# B&R Automation Studio project BRLAB12
Automation Studio 4.5.2.102

## Configuration Config1

### Task classes (Cpu.sw)
```
Cyclic#1:
  Program <- Program.prg
Binaries: udbdef, TCData, ashwd, User, asfw, arconfig, sysconf, Role, ashwac, iomap
Libraries: MotorCtrl
```

### Hardware
```
4PP065_0571_P74 : 4PP065.0571-P74 v1.1.2.0
  Connector IF5:
    ActivateDevice = 1
  ConfigurationID = firstblood_Config1
  Simulation = 1
```

## Logical view

### Library Logical/Libraries/MotorCtrl (ANSIC)

#### MotorCtrl.fun - Exported functions and function blocks
```iecst
{REDUND_ERROR} FUNCTION_BLOCK FB_Controller (*TODO: Add your comment here*) (*$GROUP=User,$CAT=User,$GROUPICON=User.png,$CATICON=User.png*)
	VAR_INPUT
		e : REAL;
	END_VAR
	VAR_OUTPUT
		u : REAL;
	END_VAR
	VAR
		k_p : REAL;
		k_i : REAL;
		iyOld : REAL;
		max_abs_value : REAL;
		dt : REAL;
		integrator : FB_Integrator;
	END_VAR
END_FUNCTION_BLOCK

{REDUND_ERROR} FUNCTION_BLOCK FB_Integrator (*TODO: Add your comment here*) (*$GROUP=User,$CAT=User,$GROUPICON=User.png,$CATICON=User.png*)
	VAR_INPUT
		in : REAL;
	END_VAR
	VAR_OUTPUT
		out : REAL;
	END_VAR
	VAR
		dt : REAL;
		temp : REAL;
	END_VAR
END_FUNCTION_BLOCK

{REDUND_ERROR} FUNCTION_BLOCK FB_Motor (*TODO: Add your comment here*) (*$GROUP=User,$CAT=User,$GROUPICON=User.png,$CATICON=User.png*)
	VAR_INPUT
		u : REAL;
	END_VAR
	VAR_OUTPUT
		w : REAL;
		phi : REAL;
	END_VAR
	VAR
		integrator1 : FB_Integrator;
		integrator2 : FB_Integrator;
		Tm : REAL;
		ke : REAL;
		dt : REAL;
	END_VAR
END_FUNCTION_BLOCK
```

#### FB_Controller.c
```c
#include <bur/plctypes.h>
#ifdef __cplusplus
	extern "C"
	{
#endif
	#include "MotorCtrl.h"
#ifdef __cplusplus
	};
#endif

void FB_Controller(struct FB_Controller* inst)
{
	// П
	double p = inst->e * inst->k_p;

	// ограничение напряжения
	if (p > inst->max_abs_value)
	{
		p = inst->max_abs_value;
	}
	else if (p < -inst->max_abs_value)
	{
		p = -inst->max_abs_value;
	}

	// И
	inst->integrator.in = inst->e * inst->k_i + inst->iyOld;
	FB_Integrator(&inst->integrator);
	double pi = p + inst->integrator.out;

	inst->u = pi;

	// ограничение выхода
	if (inst->u > inst->max_abs_value)
	{
		inst->u = inst->max_abs_value;
	}
	else if (inst->u < -inst->max_abs_value)
	{
		inst->u = -inst->max_abs_value;
	}

	// Противонакопление
	inst->iyOld = inst->u - pi;
}
```

#### FB_Integrator.c
```c
#include <bur/plctypes.h>
#ifdef __cplusplus
	extern "C"
	{
#endif
	#include "MotorCtrl.h"
#ifdef __cplusplus
	};
#endif

void FB_Integrator(struct FB_Integrator* inst)
{
	inst->temp = inst->temp + inst->in * inst->dt;
	inst->out = inst->temp;
}
```

#### FB_Motor.c
```c
#include <bur/plctypes.h>
#ifdef __cplusplus
	extern "C"
	{
#endif
	#include "MotorCtrl.h"
#ifdef __cplusplus
	};
#endif

void FB_Motor(struct FB_Motor* inst)
{
	double temp = inst->u / inst->ke - inst->w;

	inst->integrator1.in = temp / inst->Tm;
	FB_Integrator(&inst->integrator1);
	inst->w = inst->integrator1.out;

	inst->integrator2.in = inst->w;
	FB_Integrator(&inst->integrator2);
	inst->phi = inst->integrator2.out;
}
```

### Program Logical/Program

#### Variables.var
```iecst
VAR
	Controller : FB_Controller;
	Counter : UINT;
	Motor : FB_Motor;
	Speed : REAL;
	Motor2 : FB_Motor;
END_VAR
```

#### Main.c
```c
#include <bur/plctypes.h>

#ifdef _DEFAULT_INCLUDES
	#include <AsDefault.h>
#endif

void _INIT ProgramInit(void)
{
	double dt = 0.01;

	Motor.dt = dt;
	Motor.ke = 0.16;
	Motor.phi = 0;
	Motor.Tm = 0.04;
	Motor.u = 0;
	Motor.w = 0;
	Motor.integrator1.in = 0;
	Motor.integrator1.dt = dt;
	Motor.integrator1.temp = 0;
	Motor.integrator2.in = 0;
	Motor.integrator2.dt = dt;
	Motor.integrator2.temp = 0;

//	/*
	Motor2.dt = dt;
	Motor2.ke = 0.16;
	Motor2.phi = 0;
	Motor2.Tm = 0.04;
	Motor2.u = 0;
	Motor2.w = 0;
	Motor2.integrator1.in = 0;
	Motor2.integrator1.dt = dt;
	Motor2.integrator1.temp = 0;
	Motor2.integrator2.in = 0;
	Motor2.integrator2.dt = dt;
	Motor2.integrator2.temp = 0;
//	*/

	Controller.dt = dt;
	Controller.e = 0;
	Controller.iyOld = 0;
	Controller.k_i = Motor.ke;
	Controller.k_p = Motor.ke * Motor.Tm;
	Controller.max_abs_value = 12;
	Controller.integrator.in = 0;
	Controller.integrator.out = 0;
	Controller.integrator.temp = 0;
	Controller.integrator.dt = dt;

	Speed = 0;
}

void _CYCLIC ProgramCyclic(void)
{
	if(Counter == 0)
	{
		Speed = 20 - Speed;
	}
	FB_Controller(&Controller);

	Motor.u = Controller.u;
	FB_Motor(&Motor);

//	/*
	Motor2.u = Speed * Motor2.ke;
	FB_Motor(&Motor2);
//	*/

	Controller.e = Speed - Motor.w;

	Counter++;
	if(Counter == 500)
	{
		Counter = 0;
	}
}

void _EXIT ProgramExit(void)
{

}
```

Listed in the project but not available here: Logical/Libraries/MotorCtrl/Types.typ, Logical/Libraries/MotorCtrl/Constants.var
